// TIA Portal V17 export
// export: Created 2025-05-22T06:00:12.6416098Z, ExportSetting WithDefaults, DisplayName Totally Integrated Automation Portal, DisplayVersion V17 Update 8, DisplayName TIA Portal Openness, DisplayVersion V17 Update 8, DisplayName TIA Portal Version Control Interface, DisplayVersion V17, DisplayName SINAMICS Startdrive Advanced, DisplayVersion V17 SP2, DisplayName SINAMICS Startdrive G110M, G120, G120C, G120D, G120P, G115D, DisplayVersion V17 SP2, DisplayName SINAMICS Startdrive G130, G150, S120, S150, SINAMICS MV, S210, DisplayVersion V17 SP2, DisplayName STEP 7 Professional, DisplayVersion V17 Update 8, DisplayName SINUMERIK ONE STEP 7 Toolbox, DisplayVersion V17 Update 12, DisplayName SINUMERIK ONE PLC Basic Program Plus, DisplayVersion V17 Update 12, DisplayName SINUMERIK 840D sl STEP 7 Toolbox, DisplayVersion V17 Update 12, DisplayName STEP 7 Safety, DisplayVersion V17 Update 6, DisplayName WinCC Advanced, DisplayVersion V17 Update 8
FUNCTION "FC1237_UNIT_1_STATION_3_CAM_NOZZLE_CALIBRATION" : Void   // FC1237, LAD
{ S7_Optimized_Access := 'TRUE' }
VERSION : 0.1
// stored: AutoNumber false, IsIECCheckEnabled false, SetENOAutomatically false, UDAEnableTagReadback false
   VAR CONSTANT
      FC_NUMBER : DInt := 1237;
   END_VAR
   VAR_TEMP   // added for the SCL form of the ladder/FBD networks
      _w1 : Bool;
      _w2 : Bool;
   END_VAR
BEGIN

REGION Network 1: GENERAL CONDITIONS
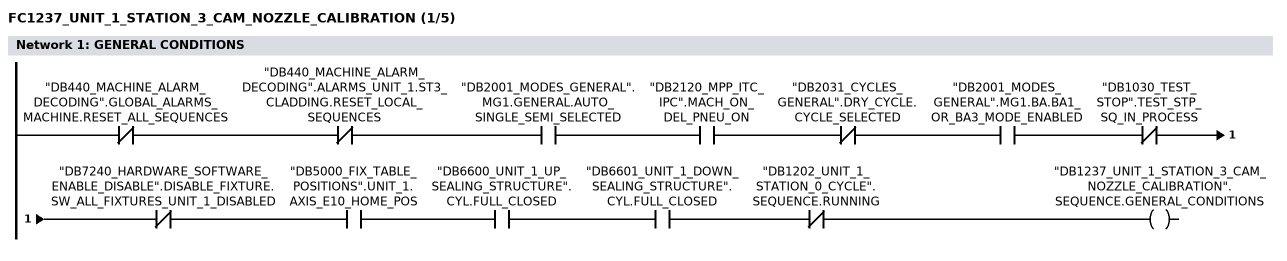
   RUNG wire#powerrail
      I_Contact( "DB440_MACHINE_ALARM_DECODING".GLOBAL_ALARMS_MACHINE.RESET_ALL_SEQUENCES )
      I_Contact( "DB440_MACHINE_ALARM_DECODING".ALARMS_UNIT_1.ST3_CLADDING.RESET_LOCAL_SEQUENCES )
      Contact( "DB2001_MODES_GENERAL".MG1.GENERAL.AUTO_SINGLE_SEMI_SELECTED )
      Contact( "DB2120_MPP_ITC_IPC".MACH_ON_DEL_PNEU_ON )
      I_Contact( "DB2031_CYCLES_GENERAL".DRY_CYCLE.CYCLE_SELECTED )
      Contact( "DB2001_MODES_GENERAL".MG1.BA.BA1_OR_BA3_MODE_ENABLED )
      I_Contact( "DB1030_TEST_STOP".TEST_STP_SQ_IN_PROCESS )
      I_Contact( "DB7240_HARDWARE_SOFTWARE_ENABLE_DISABLE".DISABLE_FIXTURE.SW_ALL_FIXTURES_UNIT_1_DISABLED )
      Contact( "DB5000_FIX_TABLE_POSITIONS".UNIT_1.AXIS_E10_HOME_POS )
      Contact( "DB6600_UNIT_1_UP_SEALING_STRUCTURE".CYL.FULL_CLOSED )
      Contact( "DB6601_UNIT_1_DOWN_SEALING_STRUCTURE".CYL.FULL_CLOSED )
      I_Contact( "DB1202_UNIT_1_STATION_0_CYCLE".SEQUENCE.RUNNING )
      Coil( "DB1237_UNIT_1_STATION_3_CAM_NOZZLE_CALIBRATION".SEQUENCE.GENERAL_CONDITIONS )
   END_RUNG
   // the same network as SCL:
   "DB1237_UNIT_1_STATION_3_CAM_NOZZLE_CALIBRATION".SEQUENCE.GENERAL_CONDITIONS := NOT "DB440_MACHINE_ALARM_DECODING".GLOBAL_ALARMS_MACHINE.RESET_ALL_SEQUENCES AND NOT "DB440_MACHINE_ALARM_DECODING".ALARMS_UNIT_1.ST3_CLADDING.RESET_LOCAL_SEQUENCES AND "DB2001_MODES_GENERAL".MG1.GENERAL.AUTO_SINGLE_SEMI_SELECTED AND "DB2120_MPP_ITC_IPC".MACH_ON_DEL_PNEU_ON AND NOT "DB2031_CYCLES_GENERAL".DRY_CYCLE.CYCLE_SELECTED AND "DB2001_MODES_GENERAL".MG1.BA.BA1_OR_BA3_MODE_ENABLED AND NOT "DB1030_TEST_STOP".TEST_STP_SQ_IN_PROCESS AND NOT "DB7240_HARDWARE_SOFTWARE_ENABLE_DISABLE".DISABLE_FIXTURE.SW_ALL_FIXTURES_UNIT_1_DISABLED AND "DB5000_FIX_TABLE_POSITIONS".UNIT_1.AXIS_E10_HOME_POS AND "DB6600_UNIT_1_UP_SEALING_STRUCTURE".CYL.FULL_CLOSED AND "DB6601_UNIT_1_DOWN_SEALING_STRUCTURE".CYL.FULL_CLOSED AND NOT "DB1202_UNIT_1_STATION_0_CYCLE".SEQUENCE.RUNNING;
END_REGION

REGION Network 2: OPERATOR HELP
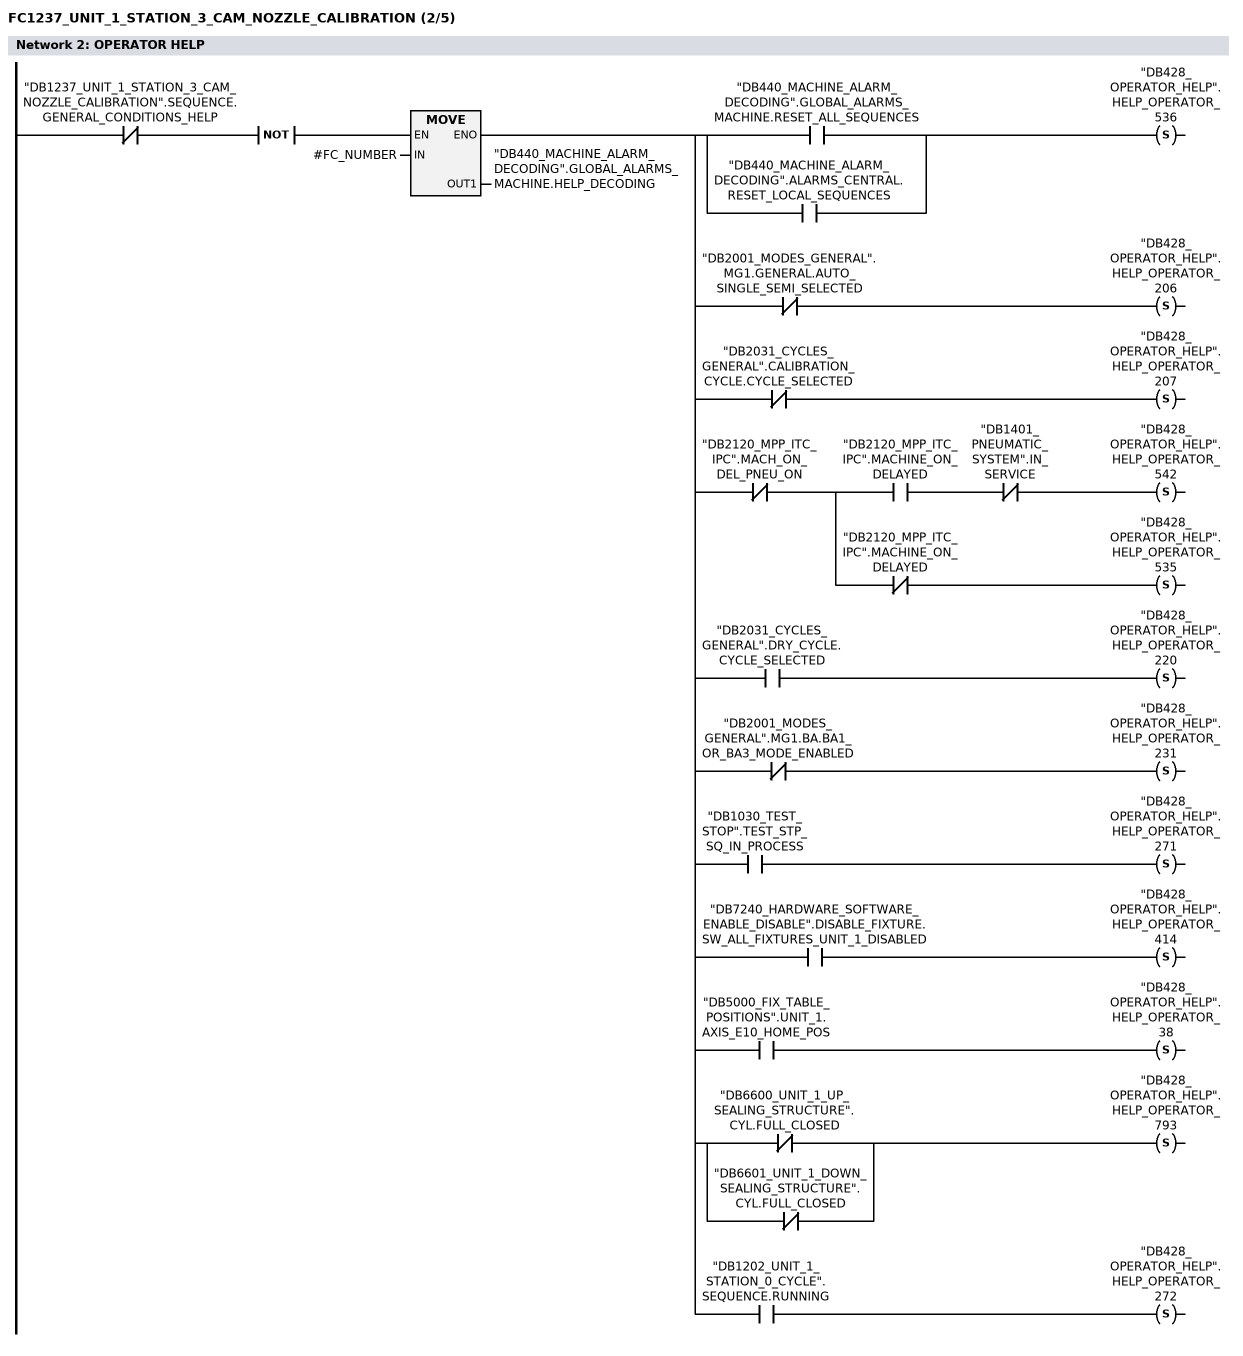
   RUNG wire#powerrail
      I_Contact( "DB1237_UNIT_1_STATION_3_CAM_NOZZLE_CALIBRATION".SEQUENCE.GENERAL_CONDITIONS_HELP )
      Not()
      { S7_GenerateENO := "TRUE" } Move(in := #FC_NUMBER, out1 => "DB440_MACHINE_ALARM_DECODING".GLOBAL_ALARMS_MACHINE.HELP_DECODING)
      wire#w1
      Contact( "DB440_MACHINE_ALARM_DECODING".GLOBAL_ALARMS_MACHINE.RESET_ALL_SEQUENCES )
      wire#w2
      S_Coil( "DB428_OPERATOR_HELP".HELP_OPERATOR_536 )
   END_RUNG
   RUNG wire#w1
      Contact( "DB440_MACHINE_ALARM_DECODING".ALARMS_CENTRAL.RESET_LOCAL_SEQUENCES )
   END_RUNG wire#w2
   RUNG wire#w1
      I_Contact( "DB2001_MODES_GENERAL".MG1.GENERAL.AUTO_SINGLE_SEMI_SELECTED )
      S_Coil( "DB428_OPERATOR_HELP".HELP_OPERATOR_206 )
   END_RUNG
   RUNG wire#w1
      I_Contact( "DB2031_CYCLES_GENERAL".CALIBRATION_CYCLE.CYCLE_SELECTED )
      S_Coil( "DB428_OPERATOR_HELP".HELP_OPERATOR_207 )
   END_RUNG
   RUNG wire#w1
      I_Contact( "DB2120_MPP_ITC_IPC".MACH_ON_DEL_PNEU_ON )
      wire#w3
      Contact( "DB2120_MPP_ITC_IPC".MACHINE_ON_DELAYED )
      I_Contact( "DB1401_PNEUMATIC_SYSTEM".IN_SERVICE )
      S_Coil( "DB428_OPERATOR_HELP".HELP_OPERATOR_542 )
   END_RUNG
   RUNG wire#w3
      I_Contact( "DB2120_MPP_ITC_IPC".MACHINE_ON_DELAYED )
      S_Coil( "DB428_OPERATOR_HELP".HELP_OPERATOR_535 )
   END_RUNG
   RUNG wire#w1
      Contact( "DB2031_CYCLES_GENERAL".DRY_CYCLE.CYCLE_SELECTED )
      S_Coil( "DB428_OPERATOR_HELP".HELP_OPERATOR_220 )
   END_RUNG
   RUNG wire#w1
      I_Contact( "DB2001_MODES_GENERAL".MG1.BA.BA1_OR_BA3_MODE_ENABLED )
      S_Coil( "DB428_OPERATOR_HELP".HELP_OPERATOR_231 )
   END_RUNG
   RUNG wire#w1
      Contact( "DB1030_TEST_STOP".TEST_STP_SQ_IN_PROCESS )
      S_Coil( "DB428_OPERATOR_HELP".HELP_OPERATOR_271 )
   END_RUNG
   RUNG wire#w1
      Contact( "DB7240_HARDWARE_SOFTWARE_ENABLE_DISABLE".DISABLE_FIXTURE.SW_ALL_FIXTURES_UNIT_1_DISABLED )
      S_Coil( "DB428_OPERATOR_HELP".HELP_OPERATOR_414 )
   END_RUNG
   RUNG wire#w1
      Contact( "DB5000_FIX_TABLE_POSITIONS".UNIT_1.AXIS_E10_HOME_POS )
      S_Coil( "DB428_OPERATOR_HELP".HELP_OPERATOR_38 )
   END_RUNG
   RUNG wire#w1
      I_Contact( "DB6600_UNIT_1_UP_SEALING_STRUCTURE".CYL.FULL_CLOSED )
      wire#w4
      S_Coil( "DB428_OPERATOR_HELP".HELP_OPERATOR_793 )
   END_RUNG
   RUNG wire#w1
      I_Contact( "DB6601_UNIT_1_DOWN_SEALING_STRUCTURE".CYL.FULL_CLOSED )
   END_RUNG wire#w4
   RUNG wire#w1
      Contact( "DB1202_UNIT_1_STATION_0_CYCLE".SEQUENCE.RUNNING )
      S_Coil( "DB428_OPERATOR_HELP".HELP_OPERATOR_272 )
   END_RUNG
   // the same network as SCL:
   // ENO of a box is taken as its EN; it also drops when the box reports an error
   #_w1 := NOT (NOT "DB1237_UNIT_1_STATION_3_CAM_NOZZLE_CALIBRATION".SEQUENCE.GENERAL_CONDITIONS_HELP);
   IF #_w1 THEN "DB440_MACHINE_ALARM_DECODING".GLOBAL_ALARMS_MACHINE.HELP_DECODING := #FC_NUMBER; END_IF;
   IF #_w1 AND ("DB440_MACHINE_ALARM_DECODING".GLOBAL_ALARMS_MACHINE.RESET_ALL_SEQUENCES OR "DB440_MACHINE_ALARM_DECODING".ALARMS_CENTRAL.RESET_LOCAL_SEQUENCES) THEN
       "DB428_OPERATOR_HELP".HELP_OPERATOR_536 := TRUE;
   END_IF;
   IF #_w1 AND NOT "DB2001_MODES_GENERAL".MG1.GENERAL.AUTO_SINGLE_SEMI_SELECTED THEN
       "DB428_OPERATOR_HELP".HELP_OPERATOR_206 := TRUE;
   END_IF;
   IF #_w1 AND NOT "DB2031_CYCLES_GENERAL".CALIBRATION_CYCLE.CYCLE_SELECTED THEN
       "DB428_OPERATOR_HELP".HELP_OPERATOR_207 := TRUE;
   END_IF;
   #_w2 := #_w1 AND NOT "DB2120_MPP_ITC_IPC".MACH_ON_DEL_PNEU_ON;
   IF #_w2 AND "DB2120_MPP_ITC_IPC".MACHINE_ON_DELAYED AND NOT "DB1401_PNEUMATIC_SYSTEM".IN_SERVICE THEN
       "DB428_OPERATOR_HELP".HELP_OPERATOR_542 := TRUE;
   END_IF;
   IF #_w2 AND NOT "DB2120_MPP_ITC_IPC".MACHINE_ON_DELAYED THEN
       "DB428_OPERATOR_HELP".HELP_OPERATOR_535 := TRUE;
   END_IF;
   IF #_w1 AND "DB2031_CYCLES_GENERAL".DRY_CYCLE.CYCLE_SELECTED THEN
       "DB428_OPERATOR_HELP".HELP_OPERATOR_220 := TRUE;
   END_IF;
   IF #_w1 AND NOT "DB2001_MODES_GENERAL".MG1.BA.BA1_OR_BA3_MODE_ENABLED THEN
       "DB428_OPERATOR_HELP".HELP_OPERATOR_231 := TRUE;
   END_IF;
   IF #_w1 AND "DB1030_TEST_STOP".TEST_STP_SQ_IN_PROCESS THEN
       "DB428_OPERATOR_HELP".HELP_OPERATOR_271 := TRUE;
   END_IF;
   IF #_w1 AND "DB7240_HARDWARE_SOFTWARE_ENABLE_DISABLE".DISABLE_FIXTURE.SW_ALL_FIXTURES_UNIT_1_DISABLED THEN
       "DB428_OPERATOR_HELP".HELP_OPERATOR_414 := TRUE;
   END_IF;
   IF #_w1 AND "DB5000_FIX_TABLE_POSITIONS".UNIT_1.AXIS_E10_HOME_POS THEN
       "DB428_OPERATOR_HELP".HELP_OPERATOR_38 := TRUE;
   END_IF;
   IF #_w1 AND (NOT "DB6600_UNIT_1_UP_SEALING_STRUCTURE".CYL.FULL_CLOSED OR NOT "DB6601_UNIT_1_DOWN_SEALING_STRUCTURE".CYL.FULL_CLOSED) THEN
       "DB428_OPERATOR_HELP".HELP_OPERATOR_793 := TRUE;
   END_IF;
   IF #_w1 AND "DB1202_UNIT_1_STATION_0_CYCLE".SEQUENCE.RUNNING THEN
       "DB428_OPERATOR_HELP".HELP_OPERATOR_272 := TRUE;
   END_IF;
END_REGION

REGION Network 3: INITIAL CONDITIONS
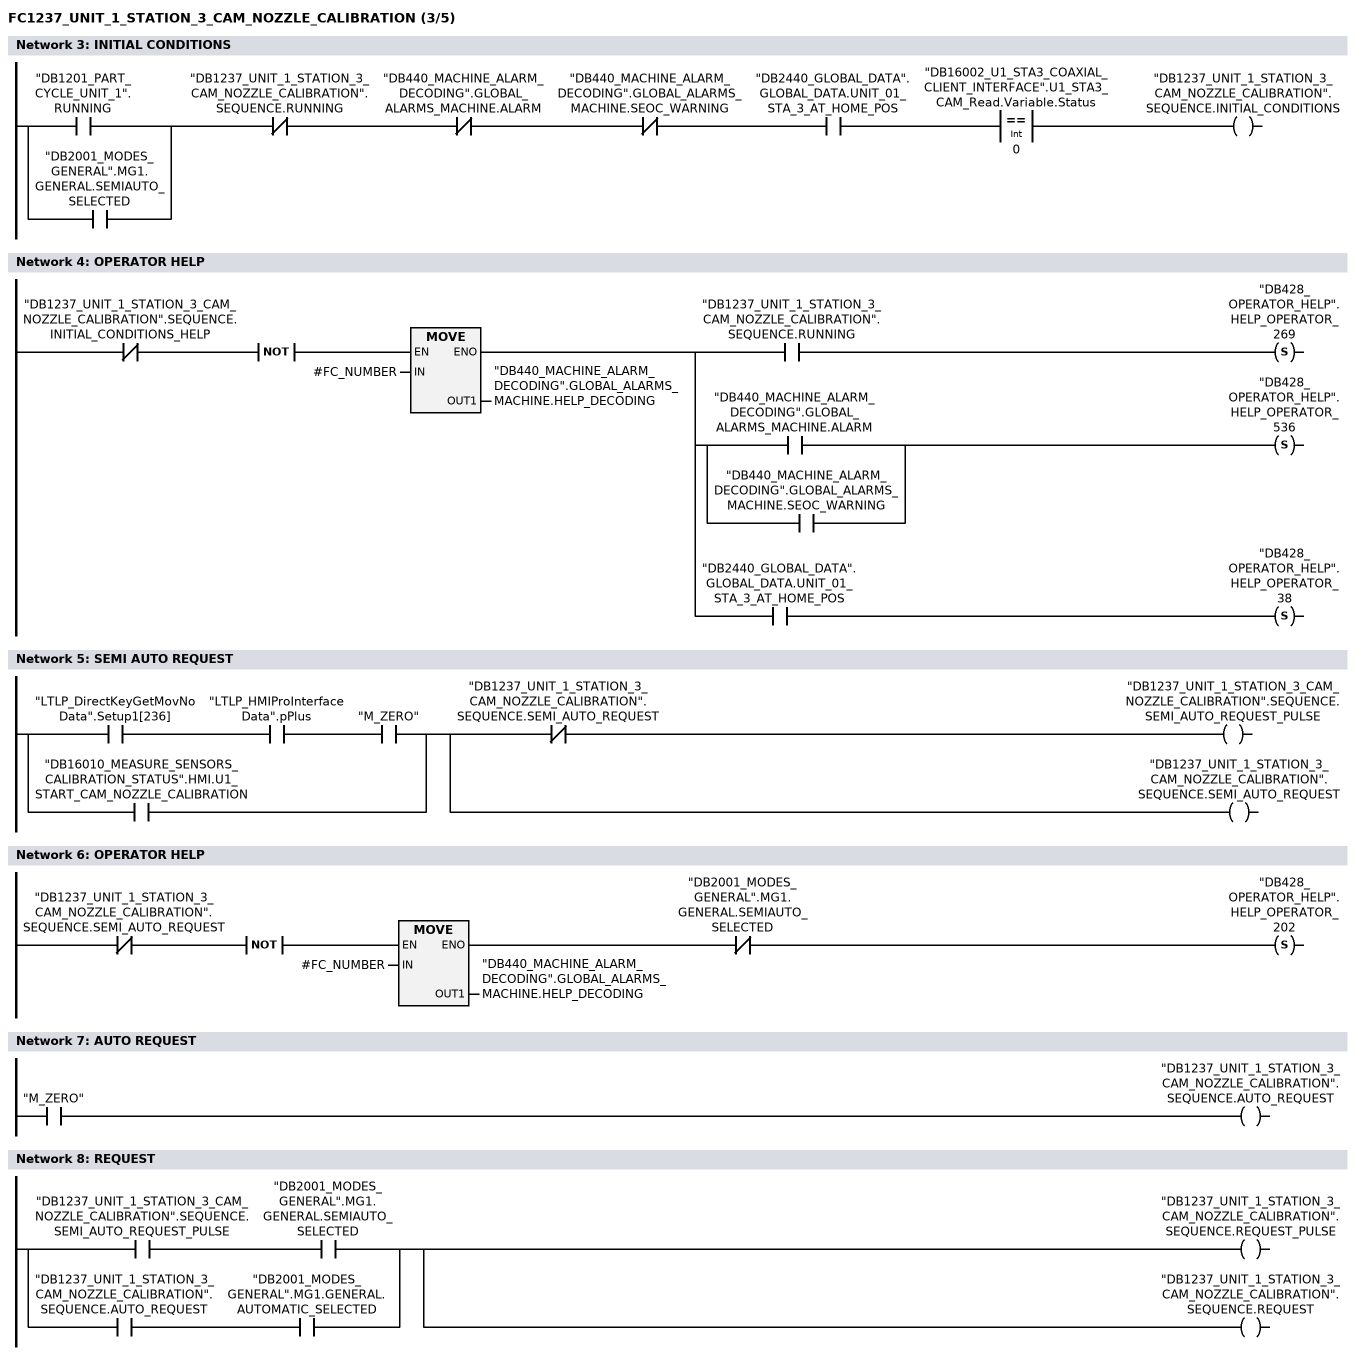
   RUNG wire#powerrail
      Contact( "DB1201_PART_CYCLE_UNIT_1".RUNNING )
      wire#w1
      I_Contact( "DB1237_UNIT_1_STATION_3_CAM_NOZZLE_CALIBRATION".SEQUENCE.RUNNING )
      I_Contact( "DB440_MACHINE_ALARM_DECODING".GLOBAL_ALARMS_MACHINE.ALARM )
      I_Contact( "DB440_MACHINE_ALARM_DECODING".GLOBAL_ALARMS_MACHINE.SEOC_WARNING )
      Contact( "DB2440_GLOBAL_DATA".GLOBAL_DATA.UNIT_01_STA_3_AT_HOME_POS )
      { S7_Templates := "SrcType := Int" } EQ_Contact(in1 := "DB16002_U1_STA3_COAXIAL_CLIENT_INTERFACE".U1_STA3_CAM_Read.Variable.Status, in2 := 0)
      Coil( "DB1237_UNIT_1_STATION_3_CAM_NOZZLE_CALIBRATION".SEQUENCE.INITIAL_CONDITIONS )
   END_RUNG
   RUNG wire#powerrail
      Contact( "DB2001_MODES_GENERAL".MG1.GENERAL.SEMIAUTO_SELECTED )
   END_RUNG wire#w1
   // the same network as SCL:
   "DB1237_UNIT_1_STATION_3_CAM_NOZZLE_CALIBRATION".SEQUENCE.INITIAL_CONDITIONS := ("DB1201_PART_CYCLE_UNIT_1".RUNNING OR "DB2001_MODES_GENERAL".MG1.GENERAL.SEMIAUTO_SELECTED) AND NOT "DB1237_UNIT_1_STATION_3_CAM_NOZZLE_CALIBRATION".SEQUENCE.RUNNING AND NOT "DB440_MACHINE_ALARM_DECODING".GLOBAL_ALARMS_MACHINE.ALARM AND NOT "DB440_MACHINE_ALARM_DECODING".GLOBAL_ALARMS_MACHINE.SEOC_WARNING AND "DB2440_GLOBAL_DATA".GLOBAL_DATA.UNIT_01_STA_3_AT_HOME_POS AND ("DB16002_U1_STA3_COAXIAL_CLIENT_INTERFACE".U1_STA3_CAM_Read.Variable.Status = 0);
END_REGION

REGION Network 4: OPERATOR HELP
   RUNG wire#powerrail
      I_Contact( "DB1237_UNIT_1_STATION_3_CAM_NOZZLE_CALIBRATION".SEQUENCE.INITIAL_CONDITIONS_HELP )
      Not()
      { S7_GenerateENO := "TRUE" } Move(in := #FC_NUMBER, out1 => "DB440_MACHINE_ALARM_DECODING".GLOBAL_ALARMS_MACHINE.HELP_DECODING)
      wire#w1
      Contact( "DB1237_UNIT_1_STATION_3_CAM_NOZZLE_CALIBRATION".SEQUENCE.RUNNING )
      S_Coil( "DB428_OPERATOR_HELP".HELP_OPERATOR_269 )
   END_RUNG
   RUNG wire#w1
      Contact( "DB440_MACHINE_ALARM_DECODING".GLOBAL_ALARMS_MACHINE.ALARM )
      wire#w2
      S_Coil( "DB428_OPERATOR_HELP".HELP_OPERATOR_536 )
   END_RUNG
   RUNG wire#w1
      Contact( "DB440_MACHINE_ALARM_DECODING".GLOBAL_ALARMS_MACHINE.SEOC_WARNING )
   END_RUNG wire#w2
   RUNG wire#w1
      Contact( "DB2440_GLOBAL_DATA".GLOBAL_DATA.UNIT_01_STA_3_AT_HOME_POS )
      S_Coil( "DB428_OPERATOR_HELP".HELP_OPERATOR_38 )
   END_RUNG
   // the same network as SCL:
   // ENO of a box is taken as its EN; it also drops when the box reports an error
   #_w1 := NOT (NOT "DB1237_UNIT_1_STATION_3_CAM_NOZZLE_CALIBRATION".SEQUENCE.INITIAL_CONDITIONS_HELP);
   IF #_w1 THEN "DB440_MACHINE_ALARM_DECODING".GLOBAL_ALARMS_MACHINE.HELP_DECODING := #FC_NUMBER; END_IF;
   IF #_w1 AND "DB1237_UNIT_1_STATION_3_CAM_NOZZLE_CALIBRATION".SEQUENCE.RUNNING THEN
       "DB428_OPERATOR_HELP".HELP_OPERATOR_269 := TRUE;
   END_IF;
   IF #_w1 AND ("DB440_MACHINE_ALARM_DECODING".GLOBAL_ALARMS_MACHINE.ALARM OR "DB440_MACHINE_ALARM_DECODING".GLOBAL_ALARMS_MACHINE.SEOC_WARNING) THEN
       "DB428_OPERATOR_HELP".HELP_OPERATOR_536 := TRUE;
   END_IF;
   IF #_w1 AND "DB2440_GLOBAL_DATA".GLOBAL_DATA.UNIT_01_STA_3_AT_HOME_POS THEN
       "DB428_OPERATOR_HELP".HELP_OPERATOR_38 := TRUE;
   END_IF;
END_REGION

REGION Network 5: SEMI AUTO REQUEST
   RUNG wire#powerrail
      Contact( "LTLP_DirectKeyGetMovNoData".Setup1[236] )
      Contact( "LTLP_HMIProInterfaceData".pPlus )
      Contact( "M_ZERO" )
      wire#w1
      I_Contact( "DB1237_UNIT_1_STATION_3_CAM_NOZZLE_CALIBRATION".SEQUENCE.SEMI_AUTO_REQUEST )
      Coil( "DB1237_UNIT_1_STATION_3_CAM_NOZZLE_CALIBRATION".SEQUENCE.SEMI_AUTO_REQUEST_PULSE )
   END_RUNG
   RUNG wire#powerrail
      Contact( "DB16010_MEASURE_SENSORS_CALIBRATION_STATUS".HMI.U1_START_CAM_NOZZLE_CALIBRATION )
   END_RUNG wire#w1
   RUNG wire#w1
      Coil( "DB1237_UNIT_1_STATION_3_CAM_NOZZLE_CALIBRATION".SEQUENCE.SEMI_AUTO_REQUEST )
   END_RUNG
   // the same network as SCL:
   #_w1 := ("LTLP_DirectKeyGetMovNoData".Setup1[236] AND "LTLP_HMIProInterfaceData".pPlus AND "M_ZERO") OR "DB16010_MEASURE_SENSORS_CALIBRATION_STATUS".HMI.U1_START_CAM_NOZZLE_CALIBRATION;
   "DB1237_UNIT_1_STATION_3_CAM_NOZZLE_CALIBRATION".SEQUENCE.SEMI_AUTO_REQUEST_PULSE := #_w1 AND NOT "DB1237_UNIT_1_STATION_3_CAM_NOZZLE_CALIBRATION".SEQUENCE.SEMI_AUTO_REQUEST;
   "DB1237_UNIT_1_STATION_3_CAM_NOZZLE_CALIBRATION".SEQUENCE.SEMI_AUTO_REQUEST := #_w1;
END_REGION

REGION Network 6: OPERATOR HELP
   RUNG wire#powerrail
      I_Contact( "DB1237_UNIT_1_STATION_3_CAM_NOZZLE_CALIBRATION".SEQUENCE.SEMI_AUTO_REQUEST )
      Not()
      { S7_GenerateENO := "TRUE" } Move(in := #FC_NUMBER, out1 => "DB440_MACHINE_ALARM_DECODING".GLOBAL_ALARMS_MACHINE.HELP_DECODING)
      I_Contact( "DB2001_MODES_GENERAL".MG1.GENERAL.SEMIAUTO_SELECTED )
      S_Coil( "DB428_OPERATOR_HELP".HELP_OPERATOR_202 )
   END_RUNG
   // the same network as SCL:
   // ENO of a box is taken as its EN; it also drops when the box reports an error
   #_w1 := NOT (NOT "DB1237_UNIT_1_STATION_3_CAM_NOZZLE_CALIBRATION".SEQUENCE.SEMI_AUTO_REQUEST);
   IF #_w1 THEN "DB440_MACHINE_ALARM_DECODING".GLOBAL_ALARMS_MACHINE.HELP_DECODING := #FC_NUMBER; END_IF;
   IF #_w1 AND NOT "DB2001_MODES_GENERAL".MG1.GENERAL.SEMIAUTO_SELECTED THEN
       "DB428_OPERATOR_HELP".HELP_OPERATOR_202 := TRUE;
   END_IF;
END_REGION

REGION Network 7: AUTO REQUEST
   RUNG wire#powerrail
      Contact( "M_ZERO" )
      Coil( "DB1237_UNIT_1_STATION_3_CAM_NOZZLE_CALIBRATION".SEQUENCE.AUTO_REQUEST )
   END_RUNG
   // the same network as SCL:
   "DB1237_UNIT_1_STATION_3_CAM_NOZZLE_CALIBRATION".SEQUENCE.AUTO_REQUEST := "M_ZERO";
END_REGION

REGION Network 8: REQUEST
   RUNG wire#powerrail
      Contact( "DB1237_UNIT_1_STATION_3_CAM_NOZZLE_CALIBRATION".SEQUENCE.SEMI_AUTO_REQUEST_PULSE )
      Contact( "DB2001_MODES_GENERAL".MG1.GENERAL.SEMIAUTO_SELECTED )
      wire#w1
      Coil( "DB1237_UNIT_1_STATION_3_CAM_NOZZLE_CALIBRATION".SEQUENCE.REQUEST_PULSE )
   END_RUNG
   RUNG wire#powerrail
      Contact( "DB1237_UNIT_1_STATION_3_CAM_NOZZLE_CALIBRATION".SEQUENCE.AUTO_REQUEST )
      Contact( "DB2001_MODES_GENERAL".MG1.GENERAL.AUTOMATIC_SELECTED )
   END_RUNG wire#w1
   RUNG wire#w1
      Coil( "DB1237_UNIT_1_STATION_3_CAM_NOZZLE_CALIBRATION".SEQUENCE.REQUEST )
   END_RUNG
   // the same network as SCL:
   "DB1237_UNIT_1_STATION_3_CAM_NOZZLE_CALIBRATION".SEQUENCE.REQUEST_PULSE := ("DB1237_UNIT_1_STATION_3_CAM_NOZZLE_CALIBRATION".SEQUENCE.SEMI_AUTO_REQUEST_PULSE AND "DB2001_MODES_GENERAL".MG1.GENERAL.SEMIAUTO_SELECTED) OR ("DB1237_UNIT_1_STATION_3_CAM_NOZZLE_CALIBRATION".SEQUENCE.AUTO_REQUEST AND "DB2001_MODES_GENERAL".MG1.GENERAL.AUTOMATIC_SELECTED);
   "DB1237_UNIT_1_STATION_3_CAM_NOZZLE_CALIBRATION".SEQUENCE.REQUEST := "DB1237_UNIT_1_STATION_3_CAM_NOZZLE_CALIBRATION".SEQUENCE.REQUEST_PULSE;
END_REGION

REGION Network 9: COMMAND
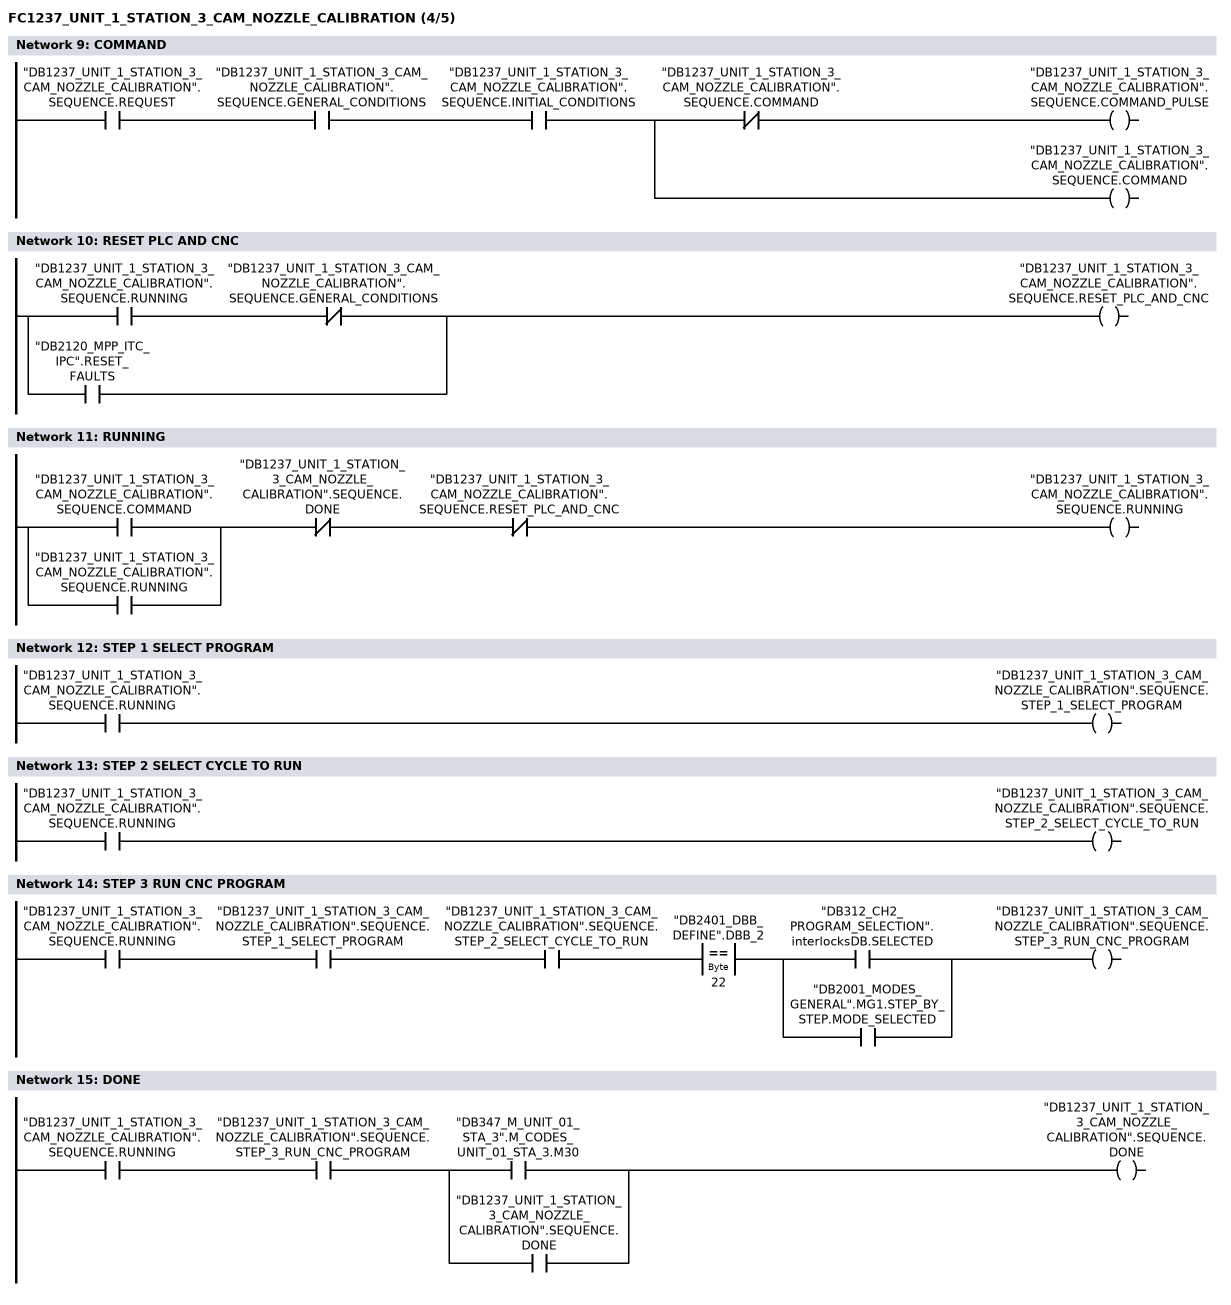
   RUNG wire#powerrail
      Contact( "DB1237_UNIT_1_STATION_3_CAM_NOZZLE_CALIBRATION".SEQUENCE.REQUEST )
      Contact( "DB1237_UNIT_1_STATION_3_CAM_NOZZLE_CALIBRATION".SEQUENCE.GENERAL_CONDITIONS )
      Contact( "DB1237_UNIT_1_STATION_3_CAM_NOZZLE_CALIBRATION".SEQUENCE.INITIAL_CONDITIONS )
      wire#w1
      I_Contact( "DB1237_UNIT_1_STATION_3_CAM_NOZZLE_CALIBRATION".SEQUENCE.COMMAND )
      Coil( "DB1237_UNIT_1_STATION_3_CAM_NOZZLE_CALIBRATION".SEQUENCE.COMMAND_PULSE )
   END_RUNG
   RUNG wire#w1
      Coil( "DB1237_UNIT_1_STATION_3_CAM_NOZZLE_CALIBRATION".SEQUENCE.COMMAND )
   END_RUNG
   // the same network as SCL:
   #_w1 := "DB1237_UNIT_1_STATION_3_CAM_NOZZLE_CALIBRATION".SEQUENCE.REQUEST AND "DB1237_UNIT_1_STATION_3_CAM_NOZZLE_CALIBRATION".SEQUENCE.GENERAL_CONDITIONS AND "DB1237_UNIT_1_STATION_3_CAM_NOZZLE_CALIBRATION".SEQUENCE.INITIAL_CONDITIONS;
   "DB1237_UNIT_1_STATION_3_CAM_NOZZLE_CALIBRATION".SEQUENCE.COMMAND_PULSE := #_w1 AND NOT "DB1237_UNIT_1_STATION_3_CAM_NOZZLE_CALIBRATION".SEQUENCE.COMMAND;
   "DB1237_UNIT_1_STATION_3_CAM_NOZZLE_CALIBRATION".SEQUENCE.COMMAND := #_w1;
END_REGION

REGION Network 10: RESET PLC AND CNC
   RUNG wire#powerrail
      Contact( "DB1237_UNIT_1_STATION_3_CAM_NOZZLE_CALIBRATION".SEQUENCE.RUNNING )
      I_Contact( "DB1237_UNIT_1_STATION_3_CAM_NOZZLE_CALIBRATION".SEQUENCE.GENERAL_CONDITIONS )
      wire#w1
      Coil( "DB1237_UNIT_1_STATION_3_CAM_NOZZLE_CALIBRATION".SEQUENCE.RESET_PLC_AND_CNC )
   END_RUNG
   RUNG wire#powerrail
      Contact( "DB2120_MPP_ITC_IPC".RESET_FAULTS )
   END_RUNG wire#w1
   // the same network as SCL:
   "DB1237_UNIT_1_STATION_3_CAM_NOZZLE_CALIBRATION".SEQUENCE.RESET_PLC_AND_CNC := ("DB1237_UNIT_1_STATION_3_CAM_NOZZLE_CALIBRATION".SEQUENCE.RUNNING AND NOT "DB1237_UNIT_1_STATION_3_CAM_NOZZLE_CALIBRATION".SEQUENCE.GENERAL_CONDITIONS) OR "DB2120_MPP_ITC_IPC".RESET_FAULTS;
END_REGION

REGION Network 11: RUNNING
   RUNG wire#powerrail
      Contact( "DB1237_UNIT_1_STATION_3_CAM_NOZZLE_CALIBRATION".SEQUENCE.COMMAND )
      wire#w1
      I_Contact( "DB1237_UNIT_1_STATION_3_CAM_NOZZLE_CALIBRATION".SEQUENCE.DONE )
      I_Contact( "DB1237_UNIT_1_STATION_3_CAM_NOZZLE_CALIBRATION".SEQUENCE.RESET_PLC_AND_CNC )
      Coil( "DB1237_UNIT_1_STATION_3_CAM_NOZZLE_CALIBRATION".SEQUENCE.RUNNING )
   END_RUNG
   RUNG wire#powerrail
      Contact( "DB1237_UNIT_1_STATION_3_CAM_NOZZLE_CALIBRATION".SEQUENCE.RUNNING )
   END_RUNG wire#w1
   // the same network as SCL:
   "DB1237_UNIT_1_STATION_3_CAM_NOZZLE_CALIBRATION".SEQUENCE.RUNNING := ("DB1237_UNIT_1_STATION_3_CAM_NOZZLE_CALIBRATION".SEQUENCE.COMMAND OR "DB1237_UNIT_1_STATION_3_CAM_NOZZLE_CALIBRATION".SEQUENCE.RUNNING) AND NOT "DB1237_UNIT_1_STATION_3_CAM_NOZZLE_CALIBRATION".SEQUENCE.DONE AND NOT "DB1237_UNIT_1_STATION_3_CAM_NOZZLE_CALIBRATION".SEQUENCE.RESET_PLC_AND_CNC;
END_REGION

REGION Network 12: STEP 1 SELECT PROGRAM
   RUNG wire#powerrail
      Contact( "DB1237_UNIT_1_STATION_3_CAM_NOZZLE_CALIBRATION".SEQUENCE.RUNNING )
      Coil( "DB1237_UNIT_1_STATION_3_CAM_NOZZLE_CALIBRATION".SEQUENCE.STEP_1_SELECT_PROGRAM )
   END_RUNG
   // the same network as SCL:
   "DB1237_UNIT_1_STATION_3_CAM_NOZZLE_CALIBRATION".SEQUENCE.STEP_1_SELECT_PROGRAM := "DB1237_UNIT_1_STATION_3_CAM_NOZZLE_CALIBRATION".SEQUENCE.RUNNING;
END_REGION

REGION Network 13: STEP 2 SELECT CYCLE TO RUN
   RUNG wire#powerrail
      Contact( "DB1237_UNIT_1_STATION_3_CAM_NOZZLE_CALIBRATION".SEQUENCE.RUNNING )
      Coil( "DB1237_UNIT_1_STATION_3_CAM_NOZZLE_CALIBRATION".SEQUENCE.STEP_2_SELECT_CYCLE_TO_RUN )
   END_RUNG
   // the same network as SCL:
   "DB1237_UNIT_1_STATION_3_CAM_NOZZLE_CALIBRATION".SEQUENCE.STEP_2_SELECT_CYCLE_TO_RUN := "DB1237_UNIT_1_STATION_3_CAM_NOZZLE_CALIBRATION".SEQUENCE.RUNNING;
END_REGION

REGION Network 14: STEP 3 RUN CNC PROGRAM
   RUNG wire#powerrail
      Contact( "DB1237_UNIT_1_STATION_3_CAM_NOZZLE_CALIBRATION".SEQUENCE.RUNNING )
      Contact( "DB1237_UNIT_1_STATION_3_CAM_NOZZLE_CALIBRATION".SEQUENCE.STEP_1_SELECT_PROGRAM )
      Contact( "DB1237_UNIT_1_STATION_3_CAM_NOZZLE_CALIBRATION".SEQUENCE.STEP_2_SELECT_CYCLE_TO_RUN )
      { S7_Templates := "SrcType := Byte" } EQ_Contact(in1 := "DB2401_DBB_DEFINE".DBB_2, in2 := 22)
      wire#w1
      Contact( "DB312_CH2_PROGRAM_SELECTION".interlocksDB.SELECTED )
      wire#w2
      Coil( "DB1237_UNIT_1_STATION_3_CAM_NOZZLE_CALIBRATION".SEQUENCE.STEP_3_RUN_CNC_PROGRAM )
   END_RUNG
   RUNG wire#w1
      Contact( "DB2001_MODES_GENERAL".MG1.STEP_BY_STEP.MODE_SELECTED )
   END_RUNG wire#w2
   // the same network as SCL:
   "DB1237_UNIT_1_STATION_3_CAM_NOZZLE_CALIBRATION".SEQUENCE.STEP_3_RUN_CNC_PROGRAM := "DB1237_UNIT_1_STATION_3_CAM_NOZZLE_CALIBRATION".SEQUENCE.RUNNING AND "DB1237_UNIT_1_STATION_3_CAM_NOZZLE_CALIBRATION".SEQUENCE.STEP_1_SELECT_PROGRAM AND "DB1237_UNIT_1_STATION_3_CAM_NOZZLE_CALIBRATION".SEQUENCE.STEP_2_SELECT_CYCLE_TO_RUN AND ("DB2401_DBB_DEFINE".DBB_2 = 22) AND ("DB312_CH2_PROGRAM_SELECTION".interlocksDB.SELECTED OR "DB2001_MODES_GENERAL".MG1.STEP_BY_STEP.MODE_SELECTED);
END_REGION

REGION Network 15: DONE
   RUNG wire#powerrail
      Contact( "DB1237_UNIT_1_STATION_3_CAM_NOZZLE_CALIBRATION".SEQUENCE.RUNNING )
      Contact( "DB1237_UNIT_1_STATION_3_CAM_NOZZLE_CALIBRATION".SEQUENCE.STEP_3_RUN_CNC_PROGRAM )
      wire#w1
      Contact( "DB347_M_UNIT_01_STA_3".M_CODES_UNIT_01_STA_3.M30 )
      wire#w2
      Coil( "DB1237_UNIT_1_STATION_3_CAM_NOZZLE_CALIBRATION".SEQUENCE.DONE )
   END_RUNG
   RUNG wire#w1
      Contact( "DB1237_UNIT_1_STATION_3_CAM_NOZZLE_CALIBRATION".SEQUENCE.DONE )
   END_RUNG wire#w2
   // the same network as SCL:
   "DB1237_UNIT_1_STATION_3_CAM_NOZZLE_CALIBRATION".SEQUENCE.DONE := "DB1237_UNIT_1_STATION_3_CAM_NOZZLE_CALIBRATION".SEQUENCE.RUNNING AND "DB1237_UNIT_1_STATION_3_CAM_NOZZLE_CALIBRATION".SEQUENCE.STEP_3_RUN_CNC_PROGRAM AND ("DB347_M_UNIT_01_STA_3".M_CODES_UNIT_01_STA_3.M30 OR "DB1237_UNIT_1_STATION_3_CAM_NOZZLE_CALIBRATION".SEQUENCE.DONE);
END_REGION

REGION Network 16: TIME EXCEEDED ALARM
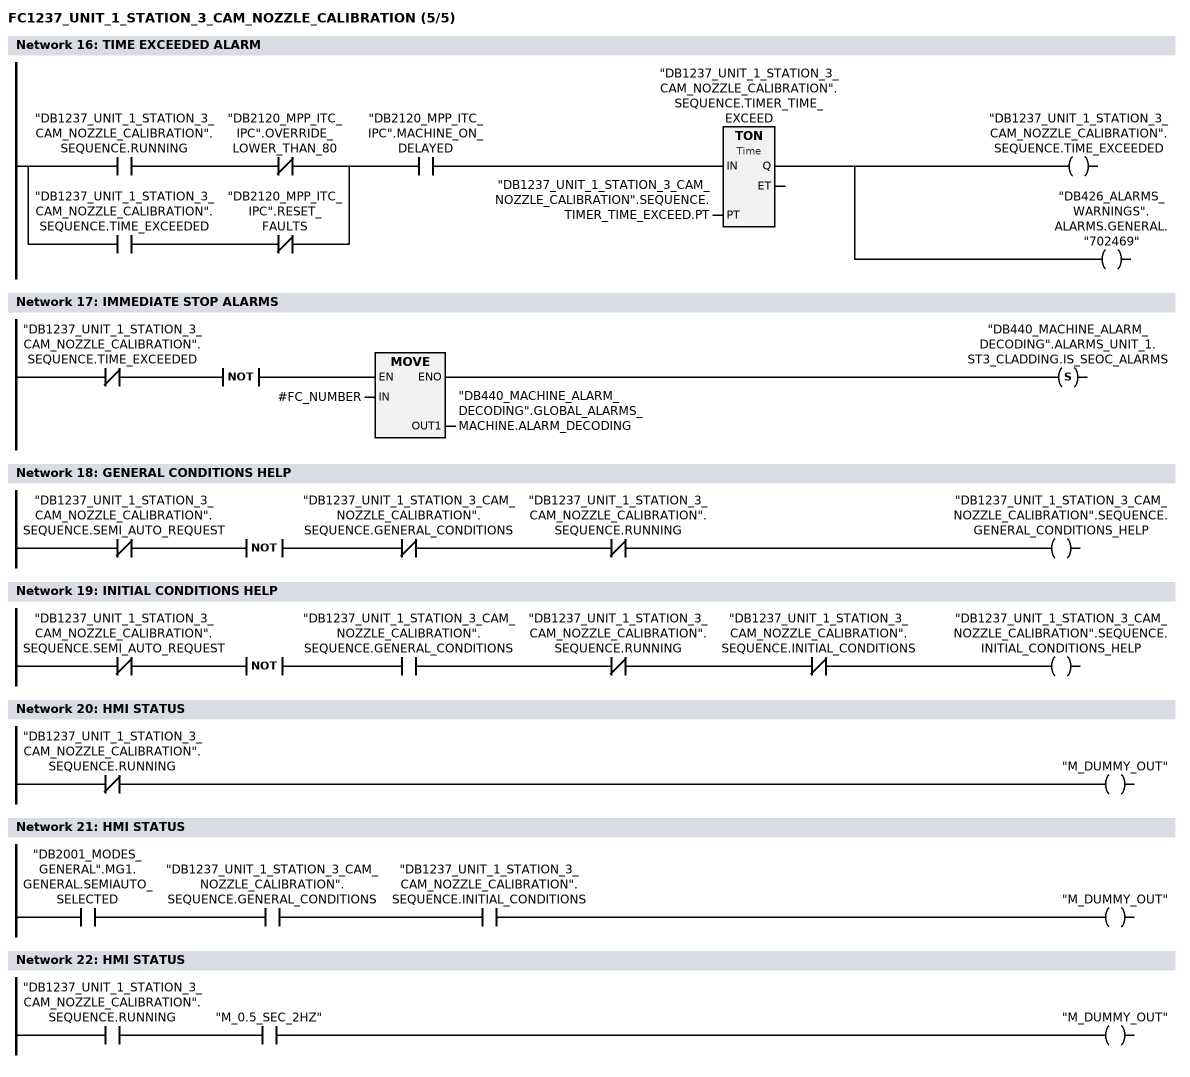
   RUNG wire#powerrail
      Contact( "DB1237_UNIT_1_STATION_3_CAM_NOZZLE_CALIBRATION".SEQUENCE.RUNNING )
      I_Contact( "DB2120_MPP_ITC_IPC".OVERRIDE_LOWER_THAN_80 )
      wire#w1
      Contact( "DB2120_MPP_ITC_IPC".MACHINE_ON_DELAYED )
      { S7_Templates := "time_type := Time" } "DB1237_UNIT_1_STATION_3_CAM_NOZZLE_CALIBRATION".SEQUENCE.TIMER_TIME_EXCEED.TON(pt := "DB1237_UNIT_1_STATION_3_CAM_NOZZLE_CALIBRATION".SEQUENCE.TIMER_TIME_EXCEED.PT, et =>)
      wire#w2
      Coil( "DB1237_UNIT_1_STATION_3_CAM_NOZZLE_CALIBRATION".SEQUENCE.TIME_EXCEEDED )
   END_RUNG
   RUNG wire#powerrail
      Contact( "DB1237_UNIT_1_STATION_3_CAM_NOZZLE_CALIBRATION".SEQUENCE.TIME_EXCEEDED )
      I_Contact( "DB2120_MPP_ITC_IPC".RESET_FAULTS )
   END_RUNG wire#w1
   RUNG wire#w2
      Coil( "DB426_ALARMS_WARNINGS".ALARMS.GENERAL."702469" )
   END_RUNG
   // the same network as SCL:
   "DB1237_UNIT_1_STATION_3_CAM_NOZZLE_CALIBRATION".SEQUENCE.TIMER_TIME_EXCEED.TON(IN := (("DB1237_UNIT_1_STATION_3_CAM_NOZZLE_CALIBRATION".SEQUENCE.RUNNING AND NOT "DB2120_MPP_ITC_IPC".OVERRIDE_LOWER_THAN_80) OR ("DB1237_UNIT_1_STATION_3_CAM_NOZZLE_CALIBRATION".SEQUENCE.TIME_EXCEEDED AND NOT "DB2120_MPP_ITC_IPC".RESET_FAULTS)) AND "DB2120_MPP_ITC_IPC".MACHINE_ON_DELAYED,
                           PT := "DB1237_UNIT_1_STATION_3_CAM_NOZZLE_CALIBRATION".SEQUENCE.TIMER_TIME_EXCEED.PT);
   "DB1237_UNIT_1_STATION_3_CAM_NOZZLE_CALIBRATION".SEQUENCE.TIME_EXCEEDED := "DB1237_UNIT_1_STATION_3_CAM_NOZZLE_CALIBRATION".SEQUENCE.TIMER_TIME_EXCEED.Q;
   "DB426_ALARMS_WARNINGS".ALARMS.GENERAL."702469" := "DB1237_UNIT_1_STATION_3_CAM_NOZZLE_CALIBRATION".SEQUENCE.TIMER_TIME_EXCEED.Q;
END_REGION

REGION Network 17: IMMEDIATE STOP ALARMS
   RUNG wire#powerrail
      I_Contact( "DB1237_UNIT_1_STATION_3_CAM_NOZZLE_CALIBRATION".SEQUENCE.TIME_EXCEEDED )
      Not()
      { S7_GenerateENO := "TRUE" } Move(in := #FC_NUMBER, out1 => "DB440_MACHINE_ALARM_DECODING".GLOBAL_ALARMS_MACHINE.ALARM_DECODING)
      S_Coil( "DB440_MACHINE_ALARM_DECODING".ALARMS_UNIT_1.ST3_CLADDING.IS_SEOC_ALARMS )
   END_RUNG
   // the same network as SCL:
   // ENO of a box is taken as its EN; it also drops when the box reports an error
   IF NOT (NOT "DB1237_UNIT_1_STATION_3_CAM_NOZZLE_CALIBRATION".SEQUENCE.TIME_EXCEEDED) THEN
       "DB440_MACHINE_ALARM_DECODING".GLOBAL_ALARMS_MACHINE.ALARM_DECODING := #FC_NUMBER;
       "DB440_MACHINE_ALARM_DECODING".ALARMS_UNIT_1.ST3_CLADDING.IS_SEOC_ALARMS := TRUE;
   END_IF;
END_REGION

REGION Network 18: GENERAL CONDITIONS HELP
   RUNG wire#powerrail
      I_Contact( "DB1237_UNIT_1_STATION_3_CAM_NOZZLE_CALIBRATION".SEQUENCE.SEMI_AUTO_REQUEST )
      Not()
      I_Contact( "DB1237_UNIT_1_STATION_3_CAM_NOZZLE_CALIBRATION".SEQUENCE.GENERAL_CONDITIONS )
      I_Contact( "DB1237_UNIT_1_STATION_3_CAM_NOZZLE_CALIBRATION".SEQUENCE.RUNNING )
      Coil( "DB1237_UNIT_1_STATION_3_CAM_NOZZLE_CALIBRATION".SEQUENCE.GENERAL_CONDITIONS_HELP )
   END_RUNG
   // the same network as SCL:
   "DB1237_UNIT_1_STATION_3_CAM_NOZZLE_CALIBRATION".SEQUENCE.GENERAL_CONDITIONS_HELP := NOT (NOT "DB1237_UNIT_1_STATION_3_CAM_NOZZLE_CALIBRATION".SEQUENCE.SEMI_AUTO_REQUEST) AND NOT "DB1237_UNIT_1_STATION_3_CAM_NOZZLE_CALIBRATION".SEQUENCE.GENERAL_CONDITIONS AND NOT "DB1237_UNIT_1_STATION_3_CAM_NOZZLE_CALIBRATION".SEQUENCE.RUNNING;
END_REGION

REGION Network 19: INITIAL CONDITIONS HELP
   RUNG wire#powerrail
      I_Contact( "DB1237_UNIT_1_STATION_3_CAM_NOZZLE_CALIBRATION".SEQUENCE.SEMI_AUTO_REQUEST )
      Not()
      Contact( "DB1237_UNIT_1_STATION_3_CAM_NOZZLE_CALIBRATION".SEQUENCE.GENERAL_CONDITIONS )
      I_Contact( "DB1237_UNIT_1_STATION_3_CAM_NOZZLE_CALIBRATION".SEQUENCE.RUNNING )
      I_Contact( "DB1237_UNIT_1_STATION_3_CAM_NOZZLE_CALIBRATION".SEQUENCE.INITIAL_CONDITIONS )
      Coil( "DB1237_UNIT_1_STATION_3_CAM_NOZZLE_CALIBRATION".SEQUENCE.INITIAL_CONDITIONS_HELP )
   END_RUNG
   // the same network as SCL:
   "DB1237_UNIT_1_STATION_3_CAM_NOZZLE_CALIBRATION".SEQUENCE.INITIAL_CONDITIONS_HELP := NOT (NOT "DB1237_UNIT_1_STATION_3_CAM_NOZZLE_CALIBRATION".SEQUENCE.SEMI_AUTO_REQUEST) AND "DB1237_UNIT_1_STATION_3_CAM_NOZZLE_CALIBRATION".SEQUENCE.GENERAL_CONDITIONS AND NOT "DB1237_UNIT_1_STATION_3_CAM_NOZZLE_CALIBRATION".SEQUENCE.RUNNING AND NOT "DB1237_UNIT_1_STATION_3_CAM_NOZZLE_CALIBRATION".SEQUENCE.INITIAL_CONDITIONS;
END_REGION

REGION Network 20: HMI STATUS
   RUNG wire#powerrail
      I_Contact( "DB1237_UNIT_1_STATION_3_CAM_NOZZLE_CALIBRATION".SEQUENCE.RUNNING )
      Coil( "M_DUMMY_OUT" )
   END_RUNG
   // the same network as SCL:
   "M_DUMMY_OUT" := NOT "DB1237_UNIT_1_STATION_3_CAM_NOZZLE_CALIBRATION".SEQUENCE.RUNNING;
END_REGION

REGION Network 21: HMI STATUS
   RUNG wire#powerrail
      Contact( "DB2001_MODES_GENERAL".MG1.GENERAL.SEMIAUTO_SELECTED )
      Contact( "DB1237_UNIT_1_STATION_3_CAM_NOZZLE_CALIBRATION".SEQUENCE.GENERAL_CONDITIONS )
      Contact( "DB1237_UNIT_1_STATION_3_CAM_NOZZLE_CALIBRATION".SEQUENCE.INITIAL_CONDITIONS )
      Coil( "M_DUMMY_OUT" )
   END_RUNG
   // the same network as SCL:
   "M_DUMMY_OUT" := "DB2001_MODES_GENERAL".MG1.GENERAL.SEMIAUTO_SELECTED AND "DB1237_UNIT_1_STATION_3_CAM_NOZZLE_CALIBRATION".SEQUENCE.GENERAL_CONDITIONS AND "DB1237_UNIT_1_STATION_3_CAM_NOZZLE_CALIBRATION".SEQUENCE.INITIAL_CONDITIONS;
END_REGION

REGION Network 22: HMI STATUS
   RUNG wire#powerrail
      Contact( "DB1237_UNIT_1_STATION_3_CAM_NOZZLE_CALIBRATION".SEQUENCE.RUNNING )
      Contact( "M_0.5_SEC_2HZ" )
      Coil( "M_DUMMY_OUT" )
   END_RUNG
   // the same network as SCL:
   "M_DUMMY_OUT" := "DB1237_UNIT_1_STATION_3_CAM_NOZZLE_CALIBRATION".SEQUENCE.RUNNING AND "M_0.5_SEC_2HZ";
END_REGION
END_FUNCTION
